FUNCTION_BLOCK GenericMaterialHolder
VAR_IN_OUT
	slots : ARRAY[*] OF STRING;
	occupied : ARRAY[*] OF BOOL;
	
	hmiTable : ARRAY[*] OF MaterialSlot;
END_VAR
VAR
	numSlots : INT;
	
	test : INT;
END_VAR

IF hmiTable <> 0 THEN
	writeHmiTable();
END_IF

numSlots := TO_INT(UPPER_BOUND(slots, 1) - LOWER_BOUND(slots, 1) + 1);

//test := SIZEOF(slots);

METHOD clear : BOOL
VAR_INPUT
END_VAR
MEMSET(ADR(slots), 0, SIZEOF(slots));
END_METHOD

METHOD findSlot : BOOL
VAR_INPUT
	materialID : STRING;
END_VAR
VAR_OUTPUT
	atSlot : INT := -1;
END_VAR
VAR
	i : INT;
END_VAR
IF materialID = '' THEN
	RETURN;
END_IF

FOR i:=1 TO GVL.maxQueue BY 1 DO
	IF slots[i] = materialID THEN
		atSlot := i;
		findSlot := TRUE;
		RETURN;
	END_IF
END_FOR
END_METHOD

METHOD getSlot : STRING
VAR_INPUT
	i : DINT;
END_VAR
VAR_OUTPUT
	errorBounds : BOOL;
END_VAR
errorBounds := i < LOWER_BOUND(slots, 1) OR i > UPPER_BOUND(slots, 1);

IF errorBounds THEN
	RETURN;
END_IF

getSlot := slots[i];
END_METHOD

METHOD getSlotsAsArray : POINTER TO STRING
getSlotsAsArray := ADR(slots);
END_METHOD

METHOD isOccupied : BOOL
VAR_INPUT
	i : DINT;
END_VAR
VAR_OUTPUT
	errorBounds : BOOL;
END_VAR
errorBounds := i < LOWER_BOUND(slots, 1) OR i > UPPER_BOUND(slots, 1);

IF errorBounds THEN
	RETURN;
END_IF

isOccupied := occupied[i];
END_METHOD

METHOD setSlots : BOOL
VAR_IN_OUT
	newSlots : ARRAY[*] OF STRING;
END_VAR
VAR
	i : DINT;
	j : DINT;
END_VAR
MEMCPY(
	slots, 
	newSlots, 
	SIZEOF(STRING) * MIN(
		(1 + UPPER_BOUND(newSlots, 1) - LOWER_BOUND(newSlots, 1)),
		(1 + UPPER_BOUND(slots, 1) - LOWER_BOUND(slots, 1))
	));
END_METHOD

METHOD PRIVATE writeHmiTable : BOOL
VAR
	i : DINT;
END_VAR
FOR i:=LOWER_BOUND(hmiTable, 1) TO UPPER_BOUND(hmiTable, 1) BY 1 DO
	hmiTable[i].material := slots[i];
	hmiTable[i].occupied := occupied[i];
END_FOR
END_METHOD

END_FUNCTION_BLOCK

(* stored: Version 1.1.0.1, ProductVersion 3.1.4024.11
   POU GenericMaterialHolder: Id {b8766d7a-1d6a-4377-9cc8-53e16c54b972}, SpecialFunc None
   Folder HMI: Id {e0175151-2858-4df9-807d-10c6bd8b5349}
   Method clear: Id {0079e54a-4897-43fe-babe-0b16afa40b6d}
   Method findSlot: Id {584be88a-e8b0-4046-8e86-717c358b8f08}
   Method getSlot: Id {de92b67f-dd7e-4c53-9c6e-8ccbe92049e8}
   Method getSlotsAsArray: Id {dff81b33-35f2-4bb2-b5f5-baf2f77d8ad6}
   Method isOccupied: Id {e248ac69-fb6d-46e9-aac8-29ec13f4c904}
   Method setSlots: Id {2ad8ecf9-54a8-4b91-9a89-b2557ee7cf42}
   Method writeHmiTable: Id {f1391623-2367-48f0-8486-56e290217047} *)
